{attribute 'qualified_only'}
VAR_GLOBAL
	// Axis
	Axis: AXIS_REF;
	
	// Function blocks
	fbPowerAxis: MC_Power;
	fbMoveContinuous: MC_MoveContinuousRelative;
	
	// Parameters
	
	PowerOverride	: LREAL := 100;
	
	// Status
	
	Power 		  : ST_MC_Status;
	MoveRelative  : ST_MC_Status;
END_VAR

(* stored: Version 1.1.0.1, ProductVersion 3.1.4024.9
   GVL GVL: Id {c0ea9552-e301-414a-bab7-d38301bde674} *)
